# B&R Automation Studio project ROS_0101a (part 2)

#### JointState.h
```c
#ifndef _ROS_sensor_msgs_JointState_h
#define _ROS_sensor_msgs_JointState_h

#include <stdint.h>
#include <string.h>
#include <stdlib.h>
#include "../ros/msg.h"
#include "../std_msgs/Header.h"

namespace sensor_msgs
{

  class JointState : public ros::Msg
  {
    public:
      typedef std_msgs::Header _header_type;
      _header_type header;
      uint32_t name_length;
      typedef char* _name_type;
      _name_type st_name;
      _name_type * name;
      uint32_t position_length;
      typedef float _position_type;
      _position_type st_position;
      _position_type * position;
      uint32_t velocity_length;
      typedef float _velocity_type;
      _velocity_type st_velocity;
      _velocity_type * velocity;
      uint32_t effort_length;
      typedef float _effort_type;
      _effort_type st_effort;
      _effort_type * effort;

    JointState():
      header(),
      name_length(0), name(NULL),
      position_length(0), position(NULL),
      velocity_length(0), velocity(NULL),
      effort_length(0), effort(NULL)
    {
    }

    virtual int serialize(unsigned char *outbuffer) const
    {
      int offset = 0;
      offset += this->header.serialize(outbuffer + offset);
      *(outbuffer + offset + 0) = (this->name_length >> (8 * 0)) & 0xFF;
      *(outbuffer + offset + 1) = (this->name_length >> (8 * 1)) & 0xFF;
      *(outbuffer + offset + 2) = (this->name_length >> (8 * 2)) & 0xFF;
      *(outbuffer + offset + 3) = (this->name_length >> (8 * 3)) & 0xFF;
      offset += sizeof(this->name_length);
      for( uint32_t i = 0; i < name_length; i++){
      uint32_t length_namei = strlen(this->name[i]);
      varToArr(outbuffer + offset, length_namei);
      offset += 4;
      memcpy(outbuffer + offset, this->name[i], length_namei);
      offset += length_namei;
      }
      *(outbuffer + offset + 0) = (this->position_length >> (8 * 0)) & 0xFF;
      *(outbuffer + offset + 1) = (this->position_length >> (8 * 1)) & 0xFF;
      *(outbuffer + offset + 2) = (this->position_length >> (8 * 2)) & 0xFF;
      *(outbuffer + offset + 3) = (this->position_length >> (8 * 3)) & 0xFF;
      offset += sizeof(this->position_length);
      for( uint32_t i = 0; i < position_length; i++){
      offset += serializeAvrFloat64(outbuffer + offset, this->position[i]);
      }
      *(outbuffer + offset + 0) = (this->velocity_length >> (8 * 0)) & 0xFF;
      *(outbuffer + offset + 1) = (this->velocity_length >> (8 * 1)) & 0xFF;
      *(outbuffer + offset + 2) = (this->velocity_length >> (8 * 2)) & 0xFF;
      *(outbuffer + offset + 3) = (this->velocity_length >> (8 * 3)) & 0xFF;
      offset += sizeof(this->velocity_length);
      for( uint32_t i = 0; i < velocity_length; i++){
      offset += serializeAvrFloat64(outbuffer + offset, this->velocity[i]);
      }
      *(outbuffer + offset + 0) = (this->effort_length >> (8 * 0)) & 0xFF;
      *(outbuffer + offset + 1) = (this->effort_length >> (8 * 1)) & 0xFF;
      *(outbuffer + offset + 2) = (this->effort_length >> (8 * 2)) & 0xFF;
      *(outbuffer + offset + 3) = (this->effort_length >> (8 * 3)) & 0xFF;
      offset += sizeof(this->effort_length);
      for( uint32_t i = 0; i < effort_length; i++){
      offset += serializeAvrFloat64(outbuffer + offset, this->effort[i]);
      }
      return offset;
    }

    virtual int deserialize(unsigned char *inbuffer)
    {
      int offset = 0;
      offset += this->header.deserialize(inbuffer + offset);
      uint32_t name_lengthT = ((uint32_t) (*(inbuffer + offset)));
      name_lengthT |= ((uint32_t) (*(inbuffer + offset + 1))) << (8 * 1);
      name_lengthT |= ((uint32_t) (*(inbuffer + offset + 2))) << (8 * 2);
      name_lengthT |= ((uint32_t) (*(inbuffer + offset + 3))) << (8 * 3);
      offset += sizeof(this->name_length);
      if(name_lengthT > name_length)
        this->name = (char**)realloc(this->name, name_lengthT * sizeof(char*));
      name_length = name_lengthT;
      for( uint32_t i = 0; i < name_length; i++){
      uint32_t length_st_name;
      arrToVar(length_st_name, (inbuffer + offset));
      offset += 4;
      for(unsigned int k= offset; k< offset+length_st_name; ++k){
          inbuffer[k-1]=inbuffer[k];
      }
      inbuffer[offset+length_st_name-1]=0;
      this->st_name = (char *)(inbuffer + offset-1);
      offset += length_st_name;
        memcpy( &(this->name[i]), &(this->st_name), sizeof(char*));
      }
      uint32_t position_lengthT = ((uint32_t) (*(inbuffer + offset)));
      position_lengthT |= ((uint32_t) (*(inbuffer + offset + 1))) << (8 * 1);
      position_lengthT |= ((uint32_t) (*(inbuffer + offset + 2))) << (8 * 2);
      position_lengthT |= ((uint32_t) (*(inbuffer + offset + 3))) << (8 * 3);
      offset += sizeof(this->position_length);
      if(position_lengthT > position_length)
        this->position = (float*)realloc(this->position, position_lengthT * sizeof(float));
      position_length = position_lengthT;
      for( uint32_t i = 0; i < position_length; i++){
      offset += deserializeAvrFloat64(inbuffer + offset, &(this->st_position));
        memcpy( &(this->position[i]), &(this->st_position), sizeof(float));
      }
      uint32_t velocity_lengthT = ((uint32_t) (*(inbuffer + offset)));
      velocity_lengthT |= ((uint32_t) (*(inbuffer + offset + 1))) << (8 * 1);
      velocity_lengthT |= ((uint32_t) (*(inbuffer + offset + 2))) << (8 * 2);
      velocity_lengthT |= ((uint32_t) (*(inbuffer + offset + 3))) << (8 * 3);
      offset += sizeof(this->velocity_length);
      if(velocity_lengthT > velocity_length)
        this->velocity = (float*)realloc(this->velocity, velocity_lengthT * sizeof(float));
      velocity_length = velocity_lengthT;
      for( uint32_t i = 0; i < velocity_length; i++){
      offset += deserializeAvrFloat64(inbuffer + offset, &(this->st_velocity));
        memcpy( &(this->velocity[i]), &(this->st_velocity), sizeof(float));
      }
      uint32_t effort_lengthT = ((uint32_t) (*(inbuffer + offset)));
      effort_lengthT |= ((uint32_t) (*(inbuffer + offset + 1))) << (8 * 1);
      effort_lengthT |= ((uint32_t) (*(inbuffer + offset + 2))) << (8 * 2);
      effort_lengthT |= ((uint32_t) (*(inbuffer + offset + 3))) << (8 * 3);
      offset += sizeof(this->effort_length);
      if(effort_lengthT > effort_length)
        this->effort = (float*)realloc(this->effort, effort_lengthT * sizeof(float));
      effort_length = effort_lengthT;
      for( uint32_t i = 0; i < effort_length; i++){
      offset += deserializeAvrFloat64(inbuffer + offset, &(this->st_effort));
        memcpy( &(this->effort[i]), &(this->st_effort), sizeof(float));
      }
     return offset;
    }

    const char * getType(){ return "sensor_msgs/JointState"; };
    const char * getMD5(){ return "3066dcd76a6cfaef579bd0f34173e9fd"; };

  };

}
#endif
```

#### node_handle.h
```c
/*
 * Software License Agreement (BSD License)
 *
 * Copyright (c) 2011, Willow Garage, Inc.
 * All rights reserved.
 *
 * Redistribution and use in source and binary forms, with or without
 * modification, are permitted provided that the following conditions
 * are met:
 *
 *  * Redistributions of source code must retain the above copyright
 *    notice, this list of conditions and the following disclaimer.
 *  * Redistributions in binary form must reproduce the above
 *    copyright notice, this list of conditions and the following
 *    disclaimer in the documentation and/or other materials provided
 *    with the distribution.
 *  * Neither the name of Willow Garage, Inc. nor the names of its
 *    contributors may be used to endorse or promote prducts derived
 *    from this software without specific prior written permission.
 *
 * THIS SOFTWARE IS PROVIDED BY THE COPYRIGHT HOLDERS AND CONTRIBUTORS
 * "AS IS" AND ANY EXPRESS OR IMPLIED WARRANTIES, INCLUDING, BUT NOT
 * LIMITED TO, THE IMPLIED WARRANTIES OF MERCHANTABILITY AND FITNESS
 * FOR A PARTICULAR PURPOSE ARE DISCLAIMED. IN NO EVENT SHALL THE
 * COPYRIGHT OWNER OR CONTRIBUTORS BE LIABLE FOR ANY DIRECT, INDIRECT,
 * INCIDENTAL, SPECIAL, EXEMPLARY, OR CONSEQUENTIAL DAMAGES (INCLUDING,
 * BUT NOT LIMITED TO, PROCUREMENT OF SUBSTITUTE GOODS OR SERVICES;
 * LOSS OF USE, DATA, OR PROFITS; OR BUSINESS INTERRUPTION) HOWEVER
 * CAUSED AND ON ANY THEORY OF LIABILITY, WHETHER IN CONTRACT, STRICT
 * LIABILITY, OR TORT (INCLUDING NEGLIGENCE OR OTHERWISE) ARISING IN
 * ANY WAY OUT OF THE USE OF THIS SOFTWARE, EVEN IF ADVISED OF THE
 * POSSIBILITY OF SUCH DAMAGE.
 */

#ifndef ROS_NODE_HANDLE_H_
#define ROS_NODE_HANDLE_H_

#include <stdint.h>

#include "std_msgs/Time.h"
#include "rosserial_msgs/TopicInfo.h"
#include "rosserial_msgs/Log.h"
#include "rosserial_msgs/RequestParam.h"

#include "ros/msg.h"

namespace ros
{

class NodeHandleBase_
{
public:
  virtual int publish(int id, const Msg* msg) = 0;
  virtual int spinOnce() = 0;
  virtual bool connected() = 0;
};
}

#include "ros/publisher.h"
#include "ros/subscriber.h"
#include "ros/service_server.h"
#include "ros/service_client.h"

namespace ros
{

const int SPIN_OK = 0;
const int SPIN_ERR = -1;
const int SPIN_TIMEOUT = -2;
const int SPIN_TIMEOUT2 = -3;

const uint8_t SYNC_SECONDS  = 5;
const uint8_t MODE_FIRST_FF = 0;
/*
 * The second sync byte is a protocol version. It's value is 0xff for the first
 * version of the rosserial protocol (used up to hydro), 0xfe for the second version
 * (introduced in hydro), 0xfd for the next, and so on. Its purpose is to enable
 * detection of mismatched protocol versions (e.g. hydro rosserial_python with groovy
 * rosserial_arduino. It must be changed in both this file and in
 * rosserial_python/src/rosserial_python/SerialClient.py
 */
const uint8_t MODE_PROTOCOL_VER   = 1;
const uint8_t PROTOCOL_VER1       = 0xff; // through groovy
const uint8_t PROTOCOL_VER2       = 0xfe; // in hydro
const uint8_t PROTOCOL_VER        = PROTOCOL_VER2;
const uint8_t MODE_SIZE_L         = 2;
const uint8_t MODE_SIZE_H         = 3;
const uint8_t MODE_SIZE_CHECKSUM  = 4;    // checksum for msg size received from size L and H
const uint8_t MODE_TOPIC_L        = 5;    // waiting for topic id
const uint8_t MODE_TOPIC_H        = 6;
const uint8_t MODE_MESSAGE        = 7;
const uint8_t MODE_MSG_CHECKSUM   = 8;    // checksum for msg and topic id

const uint8_t SERIAL_MSG_TIMEOUT  = 20;   // 20 milliseconds to recieve all of message data

using rosserial_msgs::TopicInfo;

/* Node Handle */
template<class Hardware,
         int MAX_SUBSCRIBERS = 25,
         int MAX_PUBLISHERS = 25,
         int INPUT_SIZE = 512,
         int OUTPUT_SIZE = 512>
class NodeHandle_ : public NodeHandleBase_
{
protected:
  Hardware hardware_;

  /* time used for syncing */
  uint32_t rt_time;

  /* used for computing current time */
  uint32_t sec_offset, nsec_offset;

  /* Spinonce maximum work timeout */
  uint32_t spin_timeout_;

  uint8_t message_in[INPUT_SIZE];
  uint8_t message_out[OUTPUT_SIZE];

  Publisher * publishers[MAX_PUBLISHERS];
  Subscriber_ * subscribers[MAX_SUBSCRIBERS];

  /*
   * Setup Functions
   */
public:
  NodeHandle_() : configured_(false)
  {

    for (unsigned int i = 0; i < MAX_PUBLISHERS; i++)
      publishers[i] = 0;

    for (unsigned int i = 0; i < MAX_SUBSCRIBERS; i++)
      subscribers[i] = 0;

    for (unsigned int i = 0; i < INPUT_SIZE; i++)
      message_in[i] = 0;

    for (unsigned int i = 0; i < OUTPUT_SIZE; i++)
      message_out[i] = 0;

    req_param_resp.ints_length = 0;
    req_param_resp.ints = NULL;
    req_param_resp.floats_length = 0;
    req_param_resp.floats = NULL;
    req_param_resp.ints_length = 0;
    req_param_resp.ints = NULL;

    spin_timeout_ = 0;
  }

  INT _recvCounter;
  INT _mode;
  INT _msgSize;
  INT _bytes;

  Hardware* getHardware()
  {
    return &hardware_;
  }

  /* Start serial, initialize buffers */
  void initNode()
  {
    hardware_.init();
    mode_ = 0;
    bytes_ = 0;
    index_ = 0;
    topic_ = 0;
  };

  /* Start a named port, which may be network server IP, initialize buffers */
  void initNode(char *portName)
  {
    hardware_.init(portName);
    mode_ = 0;
    bytes_ = 0;
    index_ = 0;
    topic_ = 0;
  };

  /**
   * @brief Sets the maximum time in millisconds that spinOnce() can work.
   * This will not effect the processing of the buffer, as spinOnce processes
   * one byte at a time. It simply sets the maximum time that one call can
   * process for. You can choose to clear the buffer if that is beneficial if
   * SPIN_TIMEOUT is returned from spinOnce().
   * @param timeout The timeout in milliseconds that spinOnce will function.
   */
  void setSpinTimeout(const uint32_t& timeout)
  {
     spin_timeout_ = timeout;
  }

protected:
  //State machine variables for spinOnce
  int mode_;
  int bytes_;
  int topic_;
  int index_;
  int checksum_;

  bool configured_;

  /* used for syncing the time */
  uint32_t last_sync_time;
  uint32_t last_sync_receive_time;
  uint32_t last_msg_timeout_time;

public:
  /* This function goes in your loop() function, it handles
   *  serial input and callbacks for subscribers.
   */
  virtual int spinOnce()
  {
    /* restart if timed out */
    uint32_t c_time = hardware_.time();
    if ((c_time - last_sync_receive_time) > (SYNC_SECONDS * 2200))
    {
      configured_ = false;
    }

    /* reset if message has timed out */
    if (mode_ != MODE_FIRST_FF)
    {
      if (c_time > last_msg_timeout_time)
      {
        mode_ = MODE_FIRST_FF;
      }
    }

    /* while available buffer, read data */
	while (true)
    {
	  loopCounter++;
      // If a timeout has been specified, check how long spinOnce has been running.
      if (spin_timeout_ > 0)
      {
        // If the maximum processing timeout has been exceeded, exit with error.
        // The next spinOnce can continue where it left off, or optionally
        // based on the application in use, the hardware buffer could be flushed
        // and start fresh.
        if ((hardware_.time() - c_time) > spin_timeout_)
        {
          // Exit the spin, processing timeout exceeded.
          return SPIN_TIMEOUT;
        }
      }
      int data = hardware_.read();
      if (data < 0)
        break;
      checksum_ += data;
      if (mode_ == MODE_MESSAGE)          /* message data being recieved */
      {
        message_in[index_++] = data;
        bytes_--;
        if (bytes_ == 0)                 /* is message complete? if so, checksum */
          mode_ = MODE_MSG_CHECKSUM;
      }
      else if (mode_ == MODE_FIRST_FF)
      {
        if (data == 0xff)
        {
          mode_++;
          last_msg_timeout_time = c_time + SERIAL_MSG_TIMEOUT;
        }
        else if (hardware_.time() - c_time > (SYNC_SECONDS * 1000))
        {
          /* We have been stuck in spinOnce too long, return error */
          configured_ = false;
          return SPIN_TIMEOUT;
        }
      }
      else if (mode_ == MODE_PROTOCOL_VER)
      {
        if (data == PROTOCOL_VER)
        {
          mode_++;
        }
        else
        {
          mode_ = MODE_FIRST_FF;
          if (configured_ == false)
            requestSyncTime();  /* send a msg back showing our protocol version */
        }
      }
      else if (mode_ == MODE_SIZE_L)      /* bottom half of message size */
      {
        bytes_ = data;
		_msgSize = data;
        index_ = 0;
        mode_++;
        checksum_ = data;               /* first byte for calculating size checksum */
      }
      else if (mode_ == MODE_SIZE_H)      /* top half of message size */
      {
        bytes_ += data << 8;
        mode_++;
      }
      else if (mode_ == MODE_SIZE_CHECKSUM)
      {
        if ((checksum_ % 256) == 255)
          mode_++;
        else
          mode_ = MODE_FIRST_FF;          /* Abandon the frame if the msg len is wrong */
      }
      else if (mode_ == MODE_TOPIC_L)     /* bottom half of topic id */
      {
        topic_ = data;
        mode_++;
        checksum_ = data;               /* first byte included in checksum */
      }
      else if (mode_ == MODE_TOPIC_H)     /* top half of topic id */
      {
        topic_ += data << 8;
        mode_ = MODE_MESSAGE;
        if (bytes_ == 0)
          mode_ = MODE_MSG_CHECKSUM;
      }
      else if (mode_ == MODE_MSG_CHECKSUM)    /* do checksum */
      {
        mode_ = MODE_FIRST_FF;
        if ((checksum_ % 256) == 255)
        {
          if (topic_ == TopicInfo::ID_PUBLISHER)
          {
            requestSyncTime();
            negotiateTopics();
            last_sync_time = c_time;
            last_sync_receive_time = c_time;
            return SPIN_ERR;
          }
          else if (topic_ == TopicInfo::ID_TIME)
          {
            syncTime(message_in);
          }
          else if (topic_ == TopicInfo::ID_PARAMETER_REQUEST)
          {
            req_param_resp.deserialize(message_in);
            param_recieved = true;
          }
          else if (topic_ == TopicInfo::ID_TX_STOP)
          {
            configured_ = false;
          }
          else
          {
            if (subscribers[topic_ - 100])
              subscribers[topic_ - 100]->callback(message_in);
          }
        }
      }
    }

	_mode = mode_;
	_bytes = bytes_;

    /* occasionally sync time */
    if (configured_ && ((c_time - last_sync_time) > (SYNC_SECONDS * 500)))
    {
      requestSyncTime();
      last_sync_time = c_time;
    }

    return SPIN_OK;
  }

  /* Are we connected to the PC? */
  virtual bool connected()
  {
    return configured_;
  };

  /********************************************************************
   * Time functions
   */

  void requestSyncTime()
  {
    std_msgs::Time t;
    publish(TopicInfo::ID_TIME, &t);
    rt_time = hardware_.time();
  }

  void syncTime(uint8_t * data)
  {
    std_msgs::Time t;
    uint32_t offset = hardware_.time() - rt_time;

    t.deserialize(data);
    t.data.sec += offset / 1000;
    t.data.nsec += (offset % 1000) * 1000000UL;

    this->setNow(t.data);
    last_sync_receive_time = hardware_.time();
  }

  Time now()
  {
    uint32_t ms = hardware_.time();
    Time current_time;
    current_time.sec = ms / 1000 + sec_offset;
    current_time.nsec = (ms % 1000) * 1000000UL + nsec_offset;
    normalizeSecNSec(current_time.sec, current_time.nsec);
    return current_time;
  }

  void setNow(Time & new_now)
  {
    uint32_t ms = hardware_.time();
    sec_offset = new_now.sec - ms / 1000 - 1;
    nsec_offset = new_now.nsec - (ms % 1000) * 1000000UL + 1000000000UL;
    normalizeSecNSec(sec_offset, nsec_offset);
  }

  /********************************************************************
   * Topic Management
   */

  /* Register a new publisher */
  bool advertise(Publisher & p)
  {
    for (int i = 0; i < MAX_PUBLISHERS; i++)
    {
      if (publishers[i] == 0) // empty slot
      {
        publishers[i] = &p;
        p.id_ = i + 100 + MAX_SUBSCRIBERS;
        p.nh_ = this;
        return true;
      }
    }
    return false;
  }

  /* Register a new subscriber */
  template<typename SubscriberT>
  bool subscribe(SubscriberT& s)
  {
    for (int i = 0; i < MAX_SUBSCRIBERS; i++)
    {
      if (subscribers[i] == 0) // empty slot
      {
        subscribers[i] = static_cast<Subscriber_*>(&s);
        s.id_ = i + 100;
        return true;
      }
    }
    return false;
  }

  /* Register a new Service Server */
  template<typename MReq, typename MRes, typename ObjT>
  bool advertiseService(ServiceServer<MReq, MRes, ObjT>& srv)
  {
    bool v = advertise(srv.pub);
    for (int i = 0; i < MAX_SUBSCRIBERS; i++)
    {
      if (subscribers[i] == 0) // empty slot
      {
        subscribers[i] = static_cast<Subscriber_*>(&srv);
        srv.id_ = i + 100;
        return v;
      }
    }
    return false;
  }

  /* Register a new Service Client */
  template<typename MReq, typename MRes>
  bool serviceClient(ServiceClient<MReq, MRes>& srv)
  {
    bool v = advertise(srv.pub);
    for (int i = 0; i < MAX_SUBSCRIBERS; i++)
    {
      if (subscribers[i] == 0) // empty slot
      {
        subscribers[i] = static_cast<Subscriber_*>(&srv);
        srv.id_ = i + 100;
        return v;
      }
    }
    return false;
  }

  void negotiateTopics()
  {
    rosserial_msgs::TopicInfo ti;
    int i;
    for (i = 0; i < MAX_PUBLISHERS; i++)
    {
      if (publishers[i] != 0) // non-empty slot
      {
        ti.topic_id = publishers[i]->id_;
        ti.topic_name = (char *) publishers[i]->topic_;
        ti.message_type = (char *) publishers[i]->msg_->getType();
        ti.md5sum = (char *) publishers[i]->msg_->getMD5();
        ti.buffer_size = OUTPUT_SIZE;
        publish(publishers[i]->getEndpointType(), &ti);
      }
    }
    for (i = 0; i < MAX_SUBSCRIBERS; i++)
    {
      if (subscribers[i] != 0) // non-empty slot
      {
        ti.topic_id = subscribers[i]->id_;
        ti.topic_name = (char *) subscribers[i]->topic_;
        ti.message_type = (char *) subscribers[i]->getMsgType();
        ti.md5sum = (char *) subscribers[i]->getMsgMD5();
        ti.buffer_size = INPUT_SIZE;
        publish(subscribers[i]->getEndpointType(), &ti);
      }
    }
    configured_ = true;
  }

  virtual int publish(int id, const Msg * msg)
  {
    if (id >= 100 && !configured_)
      return 0;

    /* serialize message */
    int l = msg->serialize(message_out + 7);

    /* setup the header */
    message_out[0] = 0xff;
    message_out[1] = PROTOCOL_VER;
    message_out[2] = (uint8_t)((uint16_t)l & 255);
    message_out[3] = (uint8_t)((uint16_t)l >> 8);
    message_out[4] = 255 - ((message_out[2] + message_out[3]) % 256);
    message_out[5] = (uint8_t)((int16_t)id & 255);
    message_out[6] = (uint8_t)((int16_t)id >> 8);

    /* calculate checksum */
    int chk = 0;
    for (int i = 5; i < l + 7; i++)
      chk += message_out[i];
    l += 7;
    message_out[l++] = 255 - (chk % 256);

    if (l <= OUTPUT_SIZE)
    {
      hardware_.write(message_out, l);
      return l;
    }
    else
    {
      logerror("Message from device dropped: message larger than buffer.");
      return -1;
    }
  }

  /********************************************************************
   * Logging
   */

private:
  void log(char byte, const char * msg)
  {
    rosserial_msgs::Log l;
    l.level = byte;
    l.msg = (char*)msg;
    publish(rosserial_msgs::TopicInfo::ID_LOG, &l);
  }

public:
  void logdebug(const char* msg)
  {
    log(rosserial_msgs::Log::ROSDEBUG, msg);
  }
  void loginfo(const char * msg)
  {
    log(rosserial_msgs::Log::INFO, msg);
  }
  void logwarn(const char *msg)
  {
    log(rosserial_msgs::Log::WARN, msg);
  }
  void logerror(const char*msg)
  {
    log(rosserial_msgs::Log::ERROR, msg);
  }
  void logfatal(const char*msg)
  {
    log(rosserial_msgs::Log::FATAL, msg);
  }

  /********************************************************************
   * Parameters
   */

private:
  bool param_recieved;
  rosserial_msgs::RequestParamResponse req_param_resp;

  bool requestParam(const char * name, int time_out =  1000)
  {
    param_recieved = false;
    rosserial_msgs::RequestParamRequest req;
    req.name  = (char*)name;
    publish(TopicInfo::ID_PARAMETER_REQUEST, &req);
    uint32_t end_time = hardware_.time() + time_out;
    while (!param_recieved)
    {
      spinOnce();
      if (hardware_.time() > end_time)
      {
        logwarn("Failed to get param: timeout expired");
        return false;
      }
    }
    return true;
  }

public:
  bool getParam(const char* name, int* param, int length = 1, int timeout = 1000)
  {
    if (requestParam(name, timeout))
    {
      if (length == req_param_resp.ints_length)
      {
        //copy it over
        for (int i = 0; i < length; i++)
          param[i] = req_param_resp.ints[i];
        return true;
      }
      else
      {
        logwarn("Failed to get param: length mismatch");
      }
    }
    return false;
  }
  bool getParam(const char* name, float* param, int length = 1, int timeout = 1000)
  {
    if (requestParam(name, timeout))
    {
      if (length == req_param_resp.floats_length)
      {
        //copy it over
        for (int i = 0; i < length; i++)
          param[i] = req_param_resp.floats[i];
        return true;
      }
      else
      {
        logwarn("Failed to get param: length mismatch");
      }
    }
    return false;
  }
  bool getParam(const char* name, char** param, int length = 1, int timeout = 1000)
  {
    if (requestParam(name, timeout))
    {
      if (length == req_param_resp.strings_length)
      {
        //copy it over
        for (int i = 0; i < length; i++)
          strcpy(param[i], req_param_resp.strings[i]);
        return true;
      }
      else
      {
        logwarn("Failed to get param: length mismatch");
      }
    }
    return false;
  }
  bool getParam(const char* name, bool* param, int length = 1, int timeout = 1000)
  {
    if (requestParam(name, timeout))
    {
      if (length == req_param_resp.ints_length)
      {
        //copy it over
        for (int i = 0; i < length; i++)
          param[i] = req_param_resp.ints[i];
        return true;
      }
      else
      {
        logwarn("Failed to get param: length mismatch");
      }
    }
    return false;
  }
};

}

#endif
```

#### FulfilledVoiceCommand.h
```c
#ifndef _ROS_voice_interaction_robot_msgs_FulfilledVoiceCommand_h
#define _ROS_voice_interaction_robot_msgs_FulfilledVoiceCommand_h

#include <stdint.h>
#include <string.h>
#include <stdlib.h>
#include "../ros/msg.h"
#include "../diagnostic_msgs/KeyValue.h"

namespace voice_interaction_robot_msgs
{

  class FulfilledVoiceCommand : public ros::Msg
  {
    public:
      typedef const char* _intent_name_type;
      _intent_name_type intent_name;
      uint32_t slots_length;
      typedef diagnostic_msgs::KeyValue _slots_type;
      _slots_type st_slots;
      _slots_type * slots;

    FulfilledVoiceCommand():
      intent_name(""),
      slots_length(0), slots(NULL)
    {
    }

    virtual int serialize(unsigned char *outbuffer) const
    {
      int offset = 0;
      uint32_t length_intent_name = strlen(this->intent_name);
      varToArr(outbuffer + offset, length_intent_name);
      offset += 4;
      memcpy(outbuffer + offset, this->intent_name, length_intent_name);
      offset += length_intent_name;
      *(outbuffer + offset + 0) = (this->slots_length >> (8 * 0)) & 0xFF;
      *(outbuffer + offset + 1) = (this->slots_length >> (8 * 1)) & 0xFF;
      *(outbuffer + offset + 2) = (this->slots_length >> (8 * 2)) & 0xFF;
      *(outbuffer + offset + 3) = (this->slots_length >> (8 * 3)) & 0xFF;
      offset += sizeof(this->slots_length);
      for( uint32_t i = 0; i < slots_length; i++){
      offset += this->slots[i].serialize(outbuffer + offset);
      }
      return offset;
    }

    virtual int deserialize(unsigned char *inbuffer)
    {
      int offset = 0;
      uint32_t length_intent_name;
      arrToVar(length_intent_name, (inbuffer + offset));
      offset += 4;
      for(unsigned int k= offset; k< offset+length_intent_name; ++k){
          inbuffer[k-1]=inbuffer[k];
      }
      inbuffer[offset+length_intent_name-1]=0;
      this->intent_name = (char *)(inbuffer + offset-1);
      offset += length_intent_name;
      uint32_t slots_lengthT = ((uint32_t) (*(inbuffer + offset)));
      slots_lengthT |= ((uint32_t) (*(inbuffer + offset + 1))) << (8 * 1);
      slots_lengthT |= ((uint32_t) (*(inbuffer + offset + 2))) << (8 * 2);
      slots_lengthT |= ((uint32_t) (*(inbuffer + offset + 3))) << (8 * 3);
      offset += sizeof(this->slots_length);
      if(slots_lengthT > slots_length)
        this->slots = (diagnostic_msgs::KeyValue*)realloc(this->slots, slots_lengthT * sizeof(diagnostic_msgs::KeyValue));
      slots_length = slots_lengthT;
      for( uint32_t i = 0; i < slots_length; i++){
      offset += this->st_slots.deserialize(inbuffer + offset);
        memcpy( &(this->slots[i]), &(this->st_slots), sizeof(diagnostic_msgs::KeyValue));
      }
     return offset;
    }

    const char * getType(){ return "voice_interaction_robot_msgs/FulfilledVoiceCommand"; };
    const char * getMD5(){ return "ab448516856613a366c554f14df4e422"; };

  };

}
#endif
```

#### KeyValue.h
```c
#ifndef _ROS_diagnostic_msgs_KeyValue_h
#define _ROS_diagnostic_msgs_KeyValue_h

#include <stdint.h>
#include <string.h>
#include <stdlib.h>
#include "../ros/msg.h"

namespace diagnostic_msgs
{

  class KeyValue : public ros::Msg
  {
    public:
      typedef const char* _key_type;
      _key_type key;
      typedef const char* _value_type;
      _value_type value;

    KeyValue():
      key(""),
      value("")
    {
    }

    virtual int serialize(unsigned char *outbuffer) const
    {
      int offset = 0;
      uint32_t length_key = strlen(this->key);
      varToArr(outbuffer + offset, length_key);
      offset += 4;
      memcpy(outbuffer + offset, this->key, length_key);
      offset += length_key;
      uint32_t length_value = strlen(this->value);
      varToArr(outbuffer + offset, length_value);
      offset += 4;
      memcpy(outbuffer + offset, this->value, length_value);
      offset += length_value;
      return offset;
    }

    virtual int deserialize(unsigned char *inbuffer)
    {
      int offset = 0;
      uint32_t length_key;
      arrToVar(length_key, (inbuffer + offset));
      offset += 4;
      for(unsigned int k= offset; k< offset+length_key; ++k){
          inbuffer[k-1]=inbuffer[k];
      }
      inbuffer[offset+length_key-1]=0;
      this->key = (char *)(inbuffer + offset-1);
      offset += length_key;
      uint32_t length_value;
      arrToVar(length_value, (inbuffer + offset));
      offset += 4;
      for(unsigned int k= offset; k< offset+length_value; ++k){
          inbuffer[k-1]=inbuffer[k];
      }
      inbuffer[offset+length_value-1]=0;
      this->value = (char *)(inbuffer + offset-1);
      offset += length_value;
     return offset;
    }

    const char * getType(){ return "diagnostic_msgs/KeyValue"; };
    const char * getMD5(){ return "cf57fdc6617a881a88c16e768132149c"; };

  };

}
#endif
```

#### Variables.var
```iecst
VAR
	bytes : INT;
	size : INT;
	mode : INT;
	recvCounter : INT;
	spinOnce : BOOL;
	spinCounter : DINT;
	spinMultiple : BOOL;
	New_Variable : USINT;
	spinContinuous : BOOL;
	loopCounter : UDINT;
	delayCounts : UDINT := 1000;
	totalTime : TIME;
	startTime : TIME;
	Go : BOOL;
END_VAR
```

### Program Logical/Programs/rrbotctrl (IEC)

#### Variables.var
```iecst
VAR
	joint2Position : UINT;
	joint1Position : UINT;
	PositionString : STRING[80];
	joint1Transform : STRING[1000];
	joint2Transform : STRING[1000];
	totalTransform : STRING[10000];
END_VAR
VAR CONSTANT
	PI : REAL := 3.14159;
END_VAR
VAR
	RRBotJ1 : MpAxisBasic;
	RRBotJ2 : MpAxisBasic;
	OldParameters : MpAxisBasicParType;
	RRBotJ1Parameters : MpAxisBasicParType;
	RRBotJ2Parameters : MpAxisBasicParType;
END_VAR
```

#### Main.st
```iecst
PROGRAM _INIT

	RRBotJ1.Axis := ADR(gRRBotJ1);
	RRBotJ1.MpLink := ADR(gMpLinkRRBotJ1);
	RRBotJ1.Parameters := ADR(RRBotJ1Parameters);
	RRBotJ1.Enable := TRUE;

END_PROGRAM

PROGRAM _CYCLIC

	IF (RRBotJ1.Active) THEN
		RRBotJ1.Power := TRUE;
	END_IF
	IF (RRBotJ1.PowerOn) AND (NOT RRBotJ1.IsHomed) THEN
		RRBotJ1.Home := TRUE;
	END_IF
	IF (RRBotJ1Parameters.Velocity <> OldParameters.Velocity) THEN
		RRBotJ1.Update := TRUE;
	END_IF
	IF (RRBotJ1.UpdateDone) THEN
		RRBotJ1.Update := FALSE;
	END_IF

	RRBotJ1();

	joint1SetPosition := LREAL_TO_REAL((RRBotJ1.Position) * PI / 180);

	joint1ActualPosition;
	joint2ActualPosition;

	OldParameters := RRBotJ1Parameters;

	// Handling the motion of the motors
	IF (RRBotJ1.IsHomed) THEN
		// Logic to figure out where joint 1 is
		joint1Position := REAL_TO_UINT((joint1ActualPosition * 180 / PI) + 180) MOD 360;
		brsitoa(joint1Position,ADR(PositionString));
		joint1Transform := '{"select":"#joint1Group","spin":[';
		brsstrcat(ADR(joint1Transform),ADR(PositionString));
		brsstrcat(ADR(joint1Transform),ADR(',10,0]}'));
		// Logic to figure out where joint 2 is
		joint2Position := REAL_TO_UINT(joint2ActualPosition * 180 / PI) MOD 360;
		brsitoa(joint2Position,ADR(PositionString));
		joint2Transform := '{"select":"#joint2Group","spin":[';
		brsstrcat(ADR(joint2Transform),ADR(PositionString));
		brsstrcat(ADR(joint2Transform),ADR(',10,202]}'));
	ELSE
		joint1Transform := '{"select":"#joint1Group","spin":[0,10,0]}';
		joint2Transform := '{"select":"#joint2Group","spin":[0,10,202]}';
	END_IF

	// Creating the transform string from all elements
	totalTransform := '[';
	brsstrcat(ADR(totalTransform),ADR(joint1Transform));
	brsstrcat(ADR(totalTransform),ADR(','));
	brsstrcat(ADR(totalTransform),ADR(joint2Transform));
	brsstrcat(ADR(totalTransform),ADR(']'));

	joint1PositionDegrees := fmod((joint1ActualPosition * 360 / (2 * 3.14159)) + 360, 360);
	joint2PositionDegrees := fmod((joint2ActualPosition * 360 / (2 * 3.14159)) + 360, 360);

END_PROGRAM

PROGRAM _EXIT
	(* Insert code here *)

END_PROGRAM
```


- Data object Logical/gRRBotJ1obj/gRRBotJ1a (Apt) (no source held here)

- Data object Logical/gRRBotJ1obj/gRRBotJ1i (Ax) (no source held here)

### Package Logical/gRRBotJ2obj - gRRBotJ2obj

- Data object Logical/gRRBotJ2obj/gRRBotJ2a (Apt) (no source held here)

### Data object Logical/gRRBotJ2obj/gRRBotJ2i (Ax)

#### gRRBotJ2i.ax
```
InitParameter (Version=5.4.1, NcSwId=Acp10)
  ACP10AXIS_typ:
    dig_in:
      level:
        reference = ncACTIV_HI
        pos_hw_end = ncACTIV_HI
        neg_hw_end = ncACTIV_HI
        trigger1 = ncACTIV_HI
        trigger2 = ncACTIV_HI
    encoder_if:
      parameter:
        count_dir = ncSTANDARD
        scaling:
          load:
            units = 1000
            rev_motor = 1
    limit:
      parameter:
        v_pos = 10000
        v_neg = 10000
        a1_pos = 50000
        a2_pos = 50000
        a1_neg = 50000
        a2_neg = 50000
        t_jolt = 0
        t_in_pos = 0
        pos_sw_end = 2000000000
        neg_sw_end = -2000000000
        ds_warning = 500
        ds_stop = 1000
        a_stop = 1.0e30
        dv_stop = 0
        dv_stop_mode = ncOFF
    controller:
      mode = ncPOSITION
      position:
        kv = 50
        tn = 0
        t_predict = 0.0004
        t_total = 0.0004
        p_max = 1.0e30
        i_max = 0
      speed:
        kv = 2.0
        tn = 0
        t_filter = 0.0
        isq_filter1:
          type = ncOFF
          a0 = 0.0
          a1 = 0.0
          b0 = 0.0
          b1 = 0.0
          b2 = 0.0
          c0_par_id = 0
          c1_par_id = 0
        isq_filter2:
          type = ncOFF
          a0 = 0.0
          a1 = 0.0
          b0 = 0.0
          b1 = 0.0
          b2 = 0.0
          c0_par_id = 0
          c1_par_id = 0
        isq_filter3:
          type = ncOFF
          a0 = 0.0
          a1 = 0.0
          b0 = 0.0
          b1 = 0.0
          b2 = 0.0
          c0_par_id = 0
          c1_par_id = 0
      uf:
        type = ncLINEAR + ncCORRECTION
        auto_config = ncMOTOR_PAR
        u0 = 0
        un = 0
        fn = 50.0
        k_f_slip = 0
      ff:
        mode = ncSTANDARD
        torque_load = 0.0
        torque_pos = 0.0
        torque_neg = 0.0
        kv_torque = 0.0
        inertia = 0.0
        t_filter_a = 0.0
      fb:
        mode = ncSTANDARD
        speed_mix_ratio = 0.0
        speed_kv = 2.0
      model:
        mass1:
          inertia = 0
          viscous_friction = 0
        mass2:
          inertia = 0
          viscous_friction = 0
          stiffness = 0
          damping = 0
    move:
      stop:
        parameter[0]:
          decel_ramp = ncA_LIMIT
          controller = ncON
        parameter[1]:
          decel_ramp = ncA_LIMIT
          controller = ncON
        parameter[2]:
          decel_ramp = ncA_LIMIT
          controller = ncON
        parameter[3]:
          decel_ramp = ncA_LIMIT
          controller = ncON
        quickstop:
          decel_ramp = ncA_LIMIT
          t_jolt = 0
        drive_error:
          decel_ramp = ncA_LIMIT
      homing:
        parameter:
          s = 0
          v_switch = 5000
          v_trigger = 500
          a = 50000
          mode = ncDIRECT
          edge_sw = ncPOSITIVE
          start_dir = ncPOSITIVE
          trigg_dir = ncPOSITIVE
          ref_pulse = ncOFF
          fix_dir = ncOFF
          tr_s_block = 0
          torque_lim = 0
          ds_block = 0
          ds_stop = 0
      basis:
        parameter:
          v_pos = 5000
          v_neg = 5000
          a1_pos = 50000
          a2_pos = 50000
          a1_neg = 50000
          a2_neg = 50000
    message:
      text:
        parameter:
          format = ncBREAK
          columns = 80
          data_modul = acp10etxen
```

Listed in the project but not available here: Logical/Global.typ, Logical/Libraries/RosNode/ros/duration.h, Logical/Libraries/RosNode/ros/msg.h, Logical/Libraries/RosNode/ros/duration.cpp, Logical/Libraries/RosNode/ros/time.cpp, Logical/Libraries/RosNode/rosserial_msgs/RequestMessageInfo.h, Logical/Libraries/RosNode/rosserial_msgs/RequestParam.h, Logical/Libraries/RosNode/rosserial_msgs/RequestServiceInfo.h, Logical/Libraries/RosNode/voice_interaction_robot_msgs, Logical/Libraries/RosNode/diagnostic_msgs, Logical/Programs/ros/std_msgs/Time.h, Logical/Programs/ros/std_msgs/String.h, Logical/Programs/ros/std_msgs/Float64.h, Logical/Programs/ros/ros/duration.h, Logical/Programs/ros/ros/msg.h, Logical/Programs/ros/ros/publisher.h, Logical/Programs/ros/ros/service_client.h, Logical/Programs/ros/ros/service_server.h, Logical/Programs/ros/ros/subscriber.h, Logical/Programs/ros/ros/time.h, Logical/Programs/ros/ros/duration.cpp, Logical/Programs/ros/ros/time.cpp, Logical/Programs/ros/rosserial_msgs, Logical/Programs/ros/geometry_msgs/Twist.h, Logical/Programs/ros/geometry_msgs/Vector3.h, Logical/Programs/ros/sound_play/SoundRequest.h
